INTERFACE I_Sequenceable

METHOD Execute : BOOL
END_METHOD

METHOD Reset : BOOL
END_METHOD

METHOD Abort : BOOL
END_METHOD

PROPERTY IsComplete : BOOL
GET
END_GET
END_PROPERTY

PROPERTY IsFaulted : BOOL
GET
END_GET
END_PROPERTY

PROPERTY StateName : STRING(40)
GET
END_GET
END_PROPERTY

END_INTERFACE

(* stored: Version 1.1.0.1
   Itf I_Sequenceable: Id {a1389e34-223f-4455-ab33-3d5aed9bb6d9}
   Method Execute: Id {c1f8cc95-9b08-4af9-9fc8-404fa7cafc43}
   Method Reset: Id {415e8552-6716-498f-899d-4f9399fca2db}
   Method Abort: Id {73e7e51d-5188-42bb-ba19-d4208bc1d736}
   Property IsComplete: Id {6baf7756-7931-43b3-8e45-c76877b6c151}
   Get Get: Id {728bfb1e-0be8-4019-97ec-510ea2efbd9c}
   Property IsFaulted: Id {2536a444-d47f-484b-b637-5ea0a53e8561}
   Get Get: Id {1976773f-4786-4201-baac-8932f9c6b31a}
   Property StateName: Id {17c56c01-08b8-4c64-97d1-7a1855cb36db}
   Get Get: Id {88e93306-011a-49df-8280-89e8691160f0} *)
